// Block: A0302_PareggiatoreTesta_PERS

DATA_BLOCK A0302_PareggiatoreTesta_PERS
VERSION : 0.1
   NON_RETAIN
   VAR
      Par : Struct
         Ax : Positioning_DOL_Machine_Par;
         Ax_Pers : Positioning_DOL_Machine_Pers_Data;
         Enc : PosFbk_RTN;
         Ax_Aut : A0301_Mach_Speed_Par;
         Bloccaggio_Sens : Struct
            "2111B1" : Analogic_SensorManagement_Par;
            SogliaWork : Real;
         END_STRUCT;
         CarroPareggTesta : Struct
            Delay_StartMove : Time;
            Preset : LReal;
         END_STRUCT;
         Cremaliera : Struct
            Modulo : LReal;
            Passo : LReal;
         END_STRUCT;
      END_STRUCT;
      IEC_SP : Struct
         FTC_Rall : Struct
            TON_PT : Time;
            TOF_PT : Time;
         END_STRUCT;
         FTC_ProxLs : Struct
            TON_PT : Time;
            TOF_PT : Time;
         END_STRUCT;
         FTC_PresentMat : Struct
            TON_PT : Time;
            TOF_PT : Time;
         END_STRUCT;
         Check_2111B1 : Struct
            TON_PT : Time;
         END_STRUCT;
      END_STRUCT;
   END_VAR

BEGIN
   // No initialization required
END_DATA_BLOCK
